TYPE T_Ctrl_SIf_ICL_Cur:
STRUCT
	Module: T_Ctrl_SIf_MOD_Cur;
END_STRUCT
END_TYPE

(* stored: Version 1.1.0.1, ProductVersion 3.1.0.19
   DUT T_Ctrl_SIf_ICL_Cur: Id {4b83f133-fd57-437a-ae5d-152d43a855c5} *)
